// Mitsubishi GX Works2 project: projectfinalahushiling   PLC: FX3G

// global labels: Global1
VAR_GLOBAL
  startBaking AT X001 : BOOL;
  bakingTimer AT TC6 : BOOL;
END_VAR
VAR_GLOBAL CONSTANT
  bakingSec : INT := 40;
END_VAR
VAR_GLOBAL
  endBaking AT TS6 : BOOL;
  bakingLamp AT Y004 : BOOL;
  endBakingP AT M9 : BOOL;
  startBakingTimer AT TS6 : BOOL;
  endBakingTimer AT TS6 : BOOL;
  startDay AT X010 : BOOL;
  checkStock AT M0 : BOOL;
  workDayOn AT Y010 : BOOL;
  emergancyButton AT X007 : BOOL;
  validStock AT M1 : BOOL;
  flourStock AT D1100 : REAL;
END_VAR
VAR_GLOBAL CONSTANT
  flourInit : REAL := 100;
END_VAR
VAR_GLOBAL
  flour_input AT D1150 : REAL;
  yeast_input AT D1152 : REAL;
  oil_input AT D1154 : REAL;
  water_input AT D1156 : REAL;
  spieces_input AT D1158 : REAL;
  yeastStock AT D1102 : REAL;
  oilStock AT D1104 : REAL;
  waterStock AT D1106 : REAL;
  spicesStock AT D1108 : REAL;
END_VAR
VAR_GLOBAL CONSTANT
  ratioYeast : REAL := 2.0;
  ratioOil : REAL := 3.0;
  waterRatio : REAL := 5.0;
  spicesRatio : REAL := 1.0;
  times10 : REAL := 10.0;
END_VAR
VAR_GLOBAL
  yeastTimes10 AT D1110 : REAL;
  oilTimes10 AT D1112 : REAL;
  waterTimes10 AT D1114 : REAL;
  spicesTimes10 AT D1116 : REAL;
  flourTimesYeast AT D1118 : REAL;
  flourTimesOil AT D1120 : REAL;
  flourTimesWater AT D1122 : REAL;
  flourTimesSpices AT D1124 : REAL;
  startPrep AT X002 : BOOL;
  EndPrep AT TS1 : BOOL;
  LampPrep AT Y005 : BOOL;
  timeForPrep AT TC1 : BOOL;
END_VAR
VAR_GLOBAL CONSTANT
  secondsPrep : INT := 30;
END_VAR
VAR_GLOBAL
  PrepDone AT M5 : BOOL;
END_VAR
VAR_GLOBAL CONSTANT
  yeastNeed : REAL := 20.0;
  waterNeed : REAL := 50;
  OilNeed : REAL := 30.0;
  spiceNeed : REAL := 10;
END_VAR
VAR_GLOBAL
  flourInMixer AT D1130 : REAL;
  YeastrInMixer AT D1132 : REAL;
  waterInMixer AT D1134 : REAL;
  oilInMixer AT D1136 : REAL;
  spiceInMixer AT D1138 : REAL;
  endMix AT M2 : BOOL;
  endMix2 AT M23 : BOOL;
  endMix3 AT M24 : BOOL;
  endMix4 AT M25 : BOOL;
  endMix5 AT M26 : BOOL;
  startLisha AT X001 : BOOL;
  endCountPressings AT CS0 : BOOL;
  lishaLamp AT Y001 : BOOL;
  flourInLisha AT D1140 : REAL;
  YeastrInLish AT D1142 : REAL;
  waterInLisha AT D1144 : REAL;
  oilInLisha AT D1146 : REAL;
  spiceInLisha AT D1148 : REAL;
  startSwelling AT X011 : BOOL;
END_VAR
VAR_GLOBAL CONSTANT
  doublePressings : INT := 2;
END_VAR
VAR_GLOBAL
  countPressings AT CC0 : BOOL;
  flourInProofing AT D1160 : REAL;
  YeastrInProofing AT D1162 : REAL;
  waterInProofing AT D1164 : REAL;
  oilInProofing AT D1166 : REAL;
  spiceInProofing AT D1168 : REAL;
  helpLight AT M3 : BOOL;
  flinckering2 AT Y003 : BOOL;
  flinckering1 AT Y002 : BOOL;
  TC_2 AT TC2 : BOOL;
END_VAR
VAR_GLOBAL CONSTANT
  OnOff : INT := 30;
END_VAR
VAR_GLOBAL
  TC_3 AT TC3 : BOOL;
  TS_3 AT TS3 : BOOL;
  TS_2 AT TS2 : BOOL;
  endLishaP AT M4 : BOOL;
  endProofingTimer AT TS4 : BOOL;
  proofingTimer AT TC4 : BOOL;
  endProofingP AT M4 : BOOL;
  endLisha1 AT M31 : BOOL;
  TS_4 AT TS4 : BOOL;
END_VAR
VAR_GLOBAL CONSTANT
  OnOff1 : INT := 5;
  OnOff2 : INT := 5;
END_VAR
VAR_GLOBAL
  qualityCheck AT X003 : BOOL;
  Analog_Input_2 AT D8281 : REAL;
  qualityBread AT D8201 : INT;
END_VAR
VAR_GLOBAL CONSTANT
  minQuality : INT := 400;
  maxQuality : INT := 2000;
END_VAR
VAR_GLOBAL
  startProofing AT M4 : BOOL;
  flourInBake AT D1190 : REAL;
  flourInProofingflourInBake AT D1190 : REAL;
  YeastrInBake AT D1192 : REAL;
  waterInBake AT D1194 : REAL;
  OilInBake AT D1196 : REAL;
  spiceInBake AT D1198 : REAL;
  noHaveStock AT M20 : BOOL;
  counterAnswer AT CS2 : BOOL;
  D_8281 AT D8281 : INT;
  checkCount AT CC2 : BOOL;
END_VAR
VAR_GLOBAL CONSTANT
  twoChecks : INT := 2;
END_VAR
VAR_GLOBAL
  lowThan AT M17 : BOOL;
  greaterThan AT M18 : BOOL;
  qualityCheckGood AT M11 : BOOL;
  breadReadyTimer AT TC8 : BOOL;
END_VAR
VAR_GLOBAL CONSTANT
  readyTime : INT := 50;
END_VAR
VAR_GLOBAL
  endFinishTimer AT TS8 : BOOL;
  finishLamp AT Y006 : BOOL;
  breadInBaking AT D7500 : REAL;
  breadToBakery AT D7700 : REAL;
END_VAR
VAR_GLOBAL CONSTANT
  reset : REAL;
END_VAR
VAR_GLOBAL
  dayOver AT M100 : BOOL;
  resetIngridiens AT M35 : BOOL;
  flag AT M40 : BOOL;
  Pulse AT M5 : BOOL;
  checkC AT M41 : BOOL;
  Try AT M101 : BOOL;
  reset12 AT M35 : BOOL;
  resetTry AT M50 : BOOL;
  finishLampPrep AT Y006 : BOOL;
  notEnoughIng AT M67 : BOOL;
  finishIteration AT M120 : BOOL;
  finishIteration2 AT M122 : BOOL;
  finishDay AT M20 : BOOL;
  M_51 AT M51 : BOOL;
  M_11 AT M111 : BOOL;
  M_52 AT M52 : BOOL;
  emergency AT X007 : BOOL;
  TC_7 AT TC7 : BOOL;
  TS_7 AT TS7 : BOOL;
  M_30 AT M30 : BOOL;
  TC_10 AT TC10 : BOOL;
END_VAR
VAR_GLOBAL CONSTANT
  const5 : INT := 5;
END_VAR
VAR_GLOBAL
  TS_10 AT TS10 : BOOL;
  M_12 AT M12 : BOOL;
END_VAR
VAR_GLOBAL CONSTANT
  sec3 : INT := 30;
END_VAR
VAR_GLOBAL
  TC_11 AT TC11 : BOOL;
  TS_11 AT TS11 : BOOL;
  M_111 AT M111 : BOOL;
  finishDayLight AT M20 : BOOL;
END_VAR
VAR_GLOBAL CONSTANT
  flourInit1 : REAL := 99;
END_VAR

// task Task_01 (event TRUE, interval 0, priority 31): POU_01

PROGRAM POU_01
(* structured ladder/FBD written out as ST: instructions are called as NAME(EN, inputs, outputs); _pN, _eN, _tN stand for wires *)
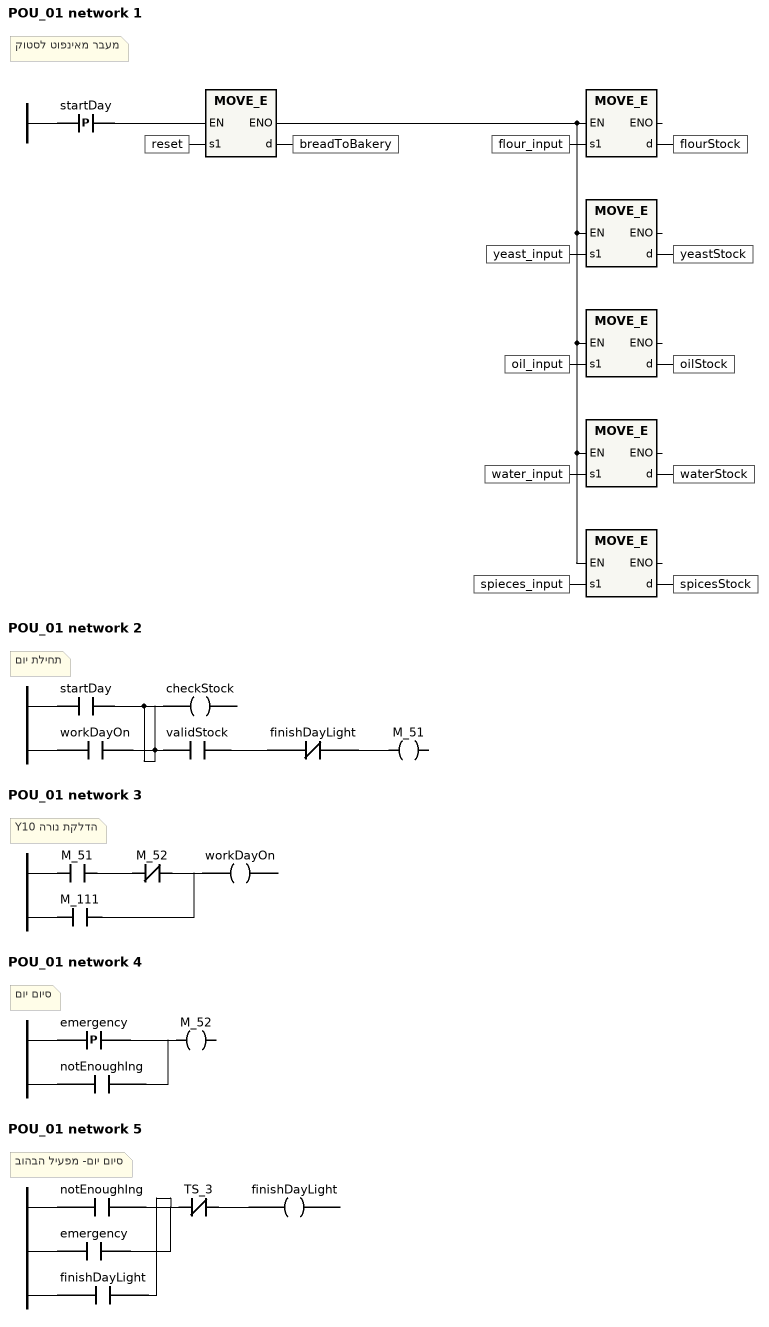
(* network 1 *)
(* מעבר מאינפוט לסטוק *)
_e1 := MOVE_E(LDP(TRUE, startDay), reset, breadToBakery);
MOVE_E(_e1, flour_input, flourStock);
MOVE_E(_e1, yeast_input, yeastStock);
MOVE_E(_e1, oil_input, oilStock);
MOVE_E(_e1, water_input, waterStock);
MOVE_E(_e1, spieces_input, spicesStock);
(* network 2 *)
(* תחילת יום *)
_p1 := startDay OR workDayOn;
checkStock := _p1;
M_51 := _p1 AND validStock AND NOT finishDayLight;
(* network 3 *)
(* הדלקת נורה Y10 *)
workDayOn := (M_51 AND NOT M_52) OR M_111;
(* network 4 *)
(* סיום יום *)
M_52 := LDP(TRUE, emergency) OR notEnoughIng;
(* network 5 *)
(* סיום יום- מפעיל הבהוב *)
finishDayLight := (notEnoughIng OR emergency OR finishDayLight) AND NOT TS_3;
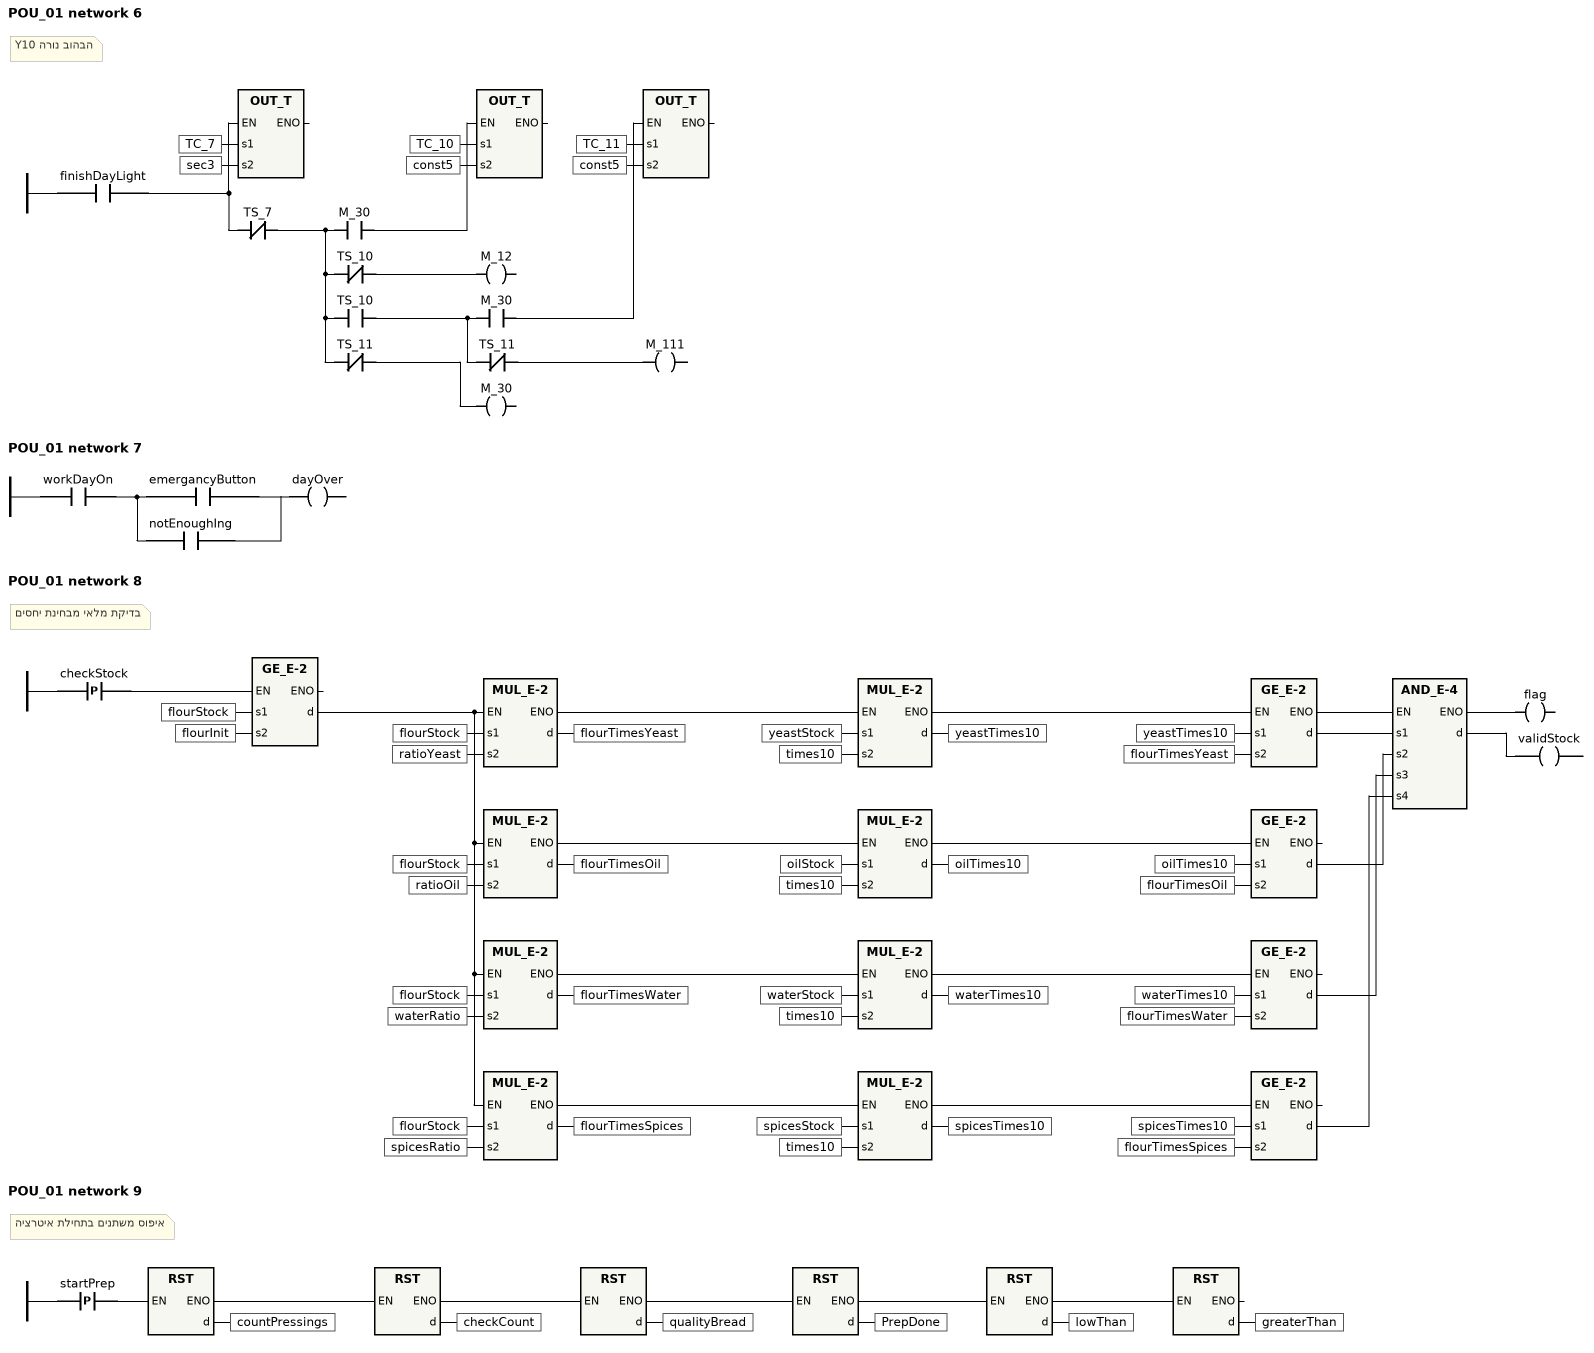
(* network 6 *)
(* הבהוב נורה Y10 *)
OUT_T(finishDayLight, TC_7, sec3);
_p1 := finishDayLight AND NOT TS_7;
OUT_T(_p1 AND M_30, TC_10, const5);
M_12 := _p1 AND NOT TS_10;
_p2 := _p1 AND TS_10;
OUT_T(_p2 AND M_30, TC_11, const5);
M_111 := _p2 AND NOT TS_11;
M_30 := _p1 AND NOT TS_11;
(* network 7 *)
dayOver := (workDayOn AND emergancyButton) OR (workDayOn AND notEnoughIng);
(* network 8 *)
(* בדיקת מלאי מבחינת יחסים *)
GE_E(LDP(TRUE, checkStock), flourStock, flourInit, _t1);
_e2 := MUL_E(_t1, flourStock, ratioYeast, flourTimesYeast);
_e3 := MUL_E(_e2, yeastStock, times10, yeastTimes10);
_e5 := GE_E(_e3, yeastTimes10, flourTimesYeast, _t4);
_e6 := MUL_E(_t1, flourStock, ratioOil, flourTimesOil);
_e7 := MUL_E(_e6, oilStock, times10, oilTimes10);
GE_E(_e7, oilTimes10, flourTimesOil, _t8);
_e9 := MUL_E(_t1, flourStock, waterRatio, flourTimesWater);
_e10 := MUL_E(_e9, waterStock, times10, waterTimes10);
GE_E(_e10, waterTimes10, flourTimesWater, _t11);
_e12 := MUL_E(_t1, flourStock, spicesRatio, flourTimesSpices);
_e13 := MUL_E(_e12, spicesStock, times10, spicesTimes10);
GE_E(_e13, spicesTimes10, flourTimesSpices, _t14);
_e16 := AND_E(_e5, _t4, _t8, _t11, _t14, _t15);
flag := _e16;
validStock := _t15;
(* network 9 *)
(* איפוס משתנים בתחילת איטרציה *)
_e1 := RST(LDP(TRUE, startPrep), countPressings);
_e2 := RST(_e1, checkCount);
_e3 := RST(_e2, qualityBread);
_e4 := RST(_e3, PrepDone);
_e5 := RST(_e4, lowThan);
RST(_e5, greaterThan);
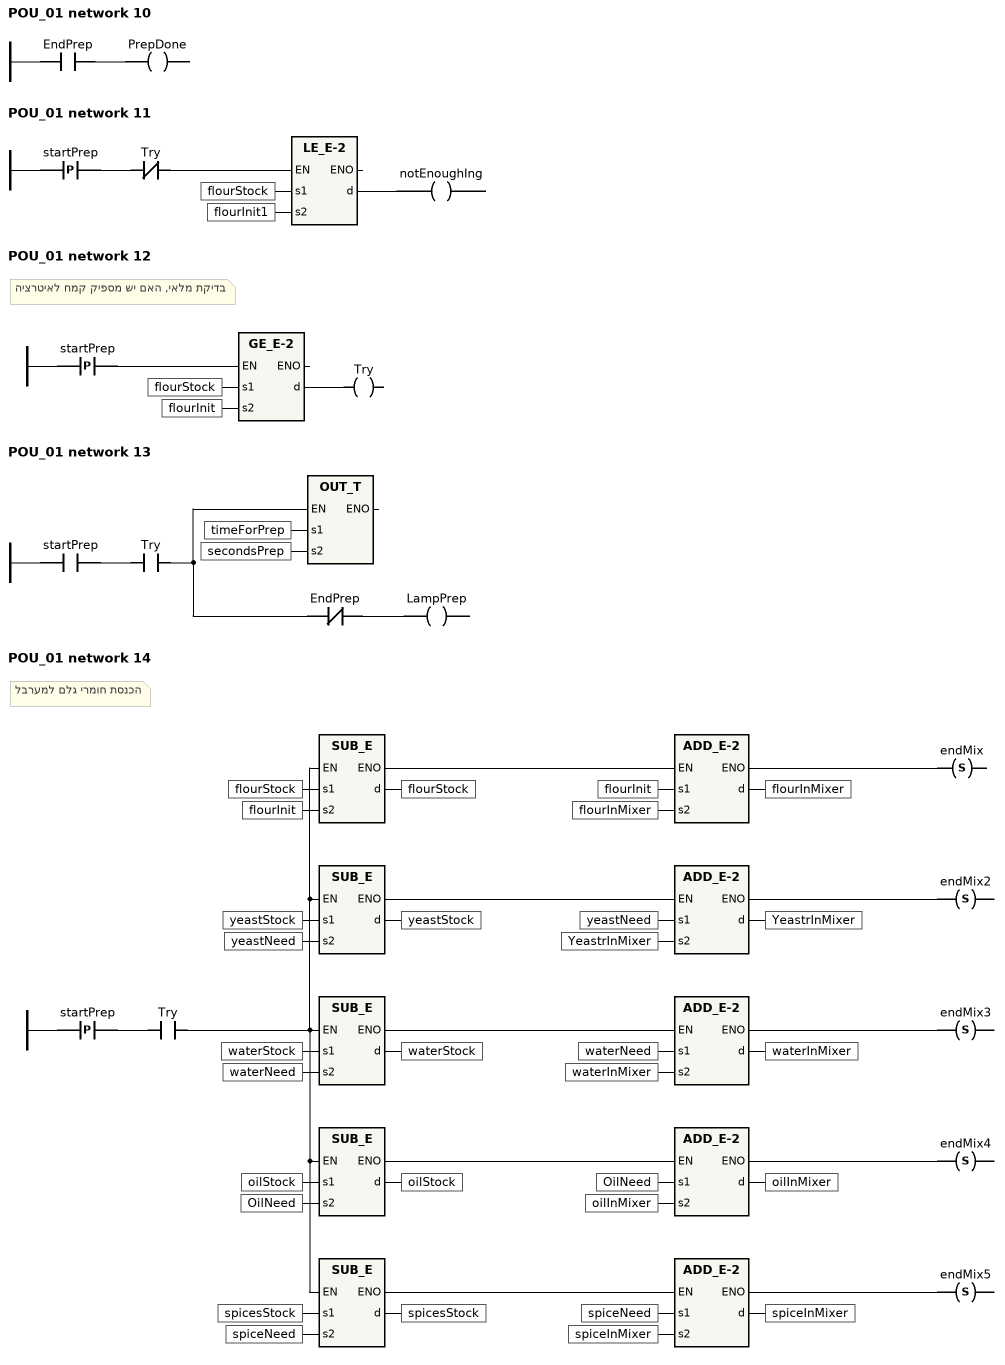
(* network 10 *)
PrepDone := EndPrep;
(* network 11 *)
LE_E(LDP(TRUE, startPrep) AND NOT Try, flourStock, flourInit1, _t1);
notEnoughIng := _t1;
(* network 12 *)
(* בדיקת מלאי, האם יש מספיק קמח לאיטרציה *)
GE_E(LDP(TRUE, startPrep), flourStock, flourInit, _t1);
Try := _t1;
(* network 13 *)
_p1 := startPrep AND Try;
OUT_T(_p1, timeForPrep, secondsPrep);
LampPrep := _p1 AND NOT EndPrep;
(* network 14 *)
(* הכנסת חומרי גלם למערבל *)
_p1 := LDP(TRUE, startPrep) AND Try;
_e2 := SUB_E(_p1, flourStock, flourInit, flourStock);
_e3 := ADD_E(_e2, flourInit, flourInMixer, flourInMixer);
SET(_e3, endMix);
_e4 := SUB_E(_p1, yeastStock, yeastNeed, yeastStock);
_e5 := ADD_E(_e4, yeastNeed, YeastrInMixer, YeastrInMixer);
SET(_e5, endMix2);
_e6 := SUB_E(_p1, waterStock, waterNeed, waterStock);
_e7 := ADD_E(_e6, waterNeed, waterInMixer, waterInMixer);
SET(_e7, endMix3);
_e8 := SUB_E(_p1, oilStock, OilNeed, oilStock);
_e9 := ADD_E(_e8, OilNeed, oilInMixer, oilInMixer);
SET(_e9, endMix4);
_e10 := SUB_E(_p1, spicesStock, spiceNeed, spicesStock);
_e11 := ADD_E(_e10, spiceNeed, spiceInMixer, spiceInMixer);
SET(_e11, endMix5);
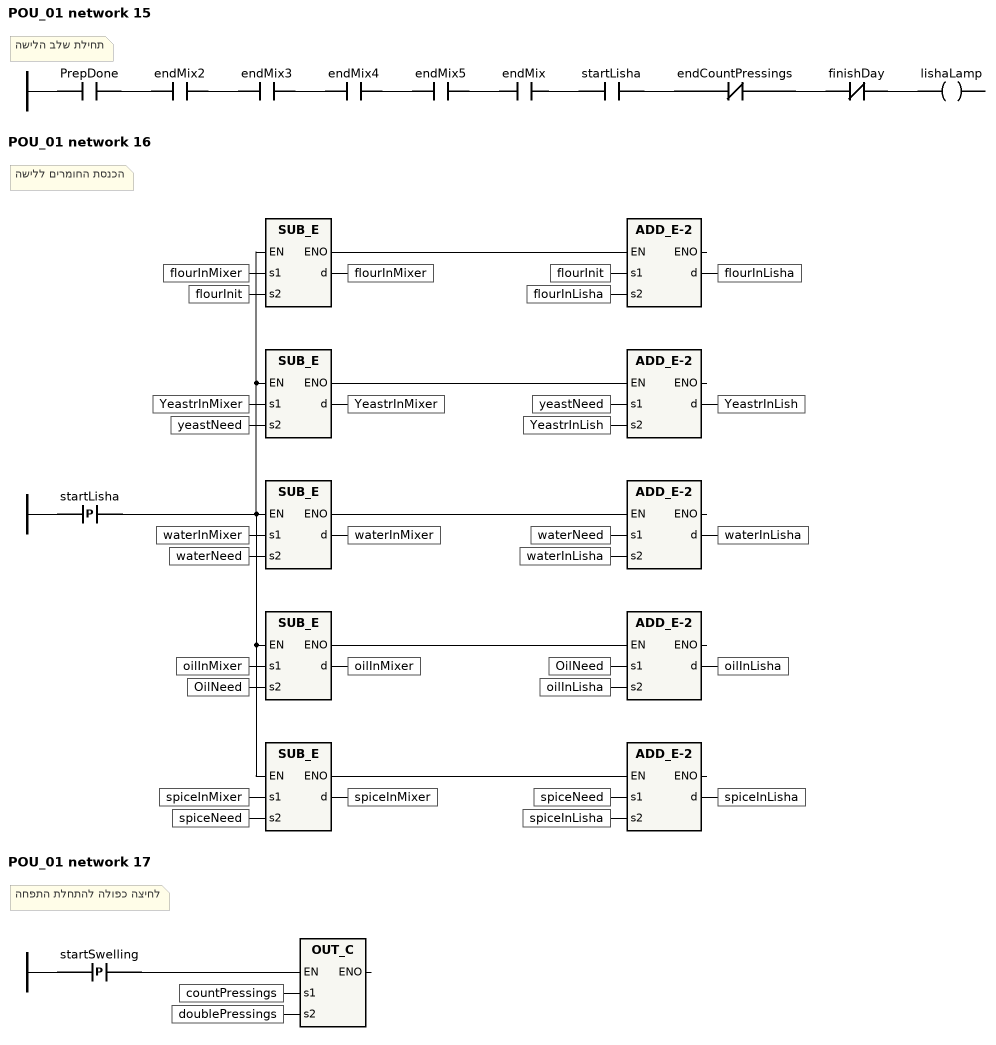
(* network 15 *)
(* תחילת שלב הלישה *)
lishaLamp := PrepDone AND endMix2 AND endMix3 AND endMix4 AND endMix5 AND endMix AND startLisha AND NOT endCountPressings AND NOT finishDay;
(* network 16 *)
(* הכנסת החומרים ללישה *)
_p1 := LDP(TRUE, startLisha);
_e2 := SUB_E(_p1, flourInMixer, flourInit, flourInMixer);
ADD_E(_e2, flourInit, flourInLisha, flourInLisha);
_e3 := SUB_E(_p1, YeastrInMixer, yeastNeed, YeastrInMixer);
ADD_E(_e3, yeastNeed, YeastrInLish, YeastrInLish);
_e4 := SUB_E(_p1, waterInMixer, waterNeed, waterInMixer);
ADD_E(_e4, waterNeed, waterInLisha, waterInLisha);
_e5 := SUB_E(_p1, oilInMixer, OilNeed, oilInMixer);
ADD_E(_e5, OilNeed, oilInLisha, oilInLisha);
_e6 := SUB_E(_p1, spiceInMixer, spiceNeed, spiceInMixer);
ADD_E(_e6, spiceNeed, spiceInLisha, spiceInLisha);
(* network 17 *)
(* לחיצה כפולה להתחלת התפחה *)
OUT_C(LDP(TRUE, startSwelling), countPressings, doublePressings);
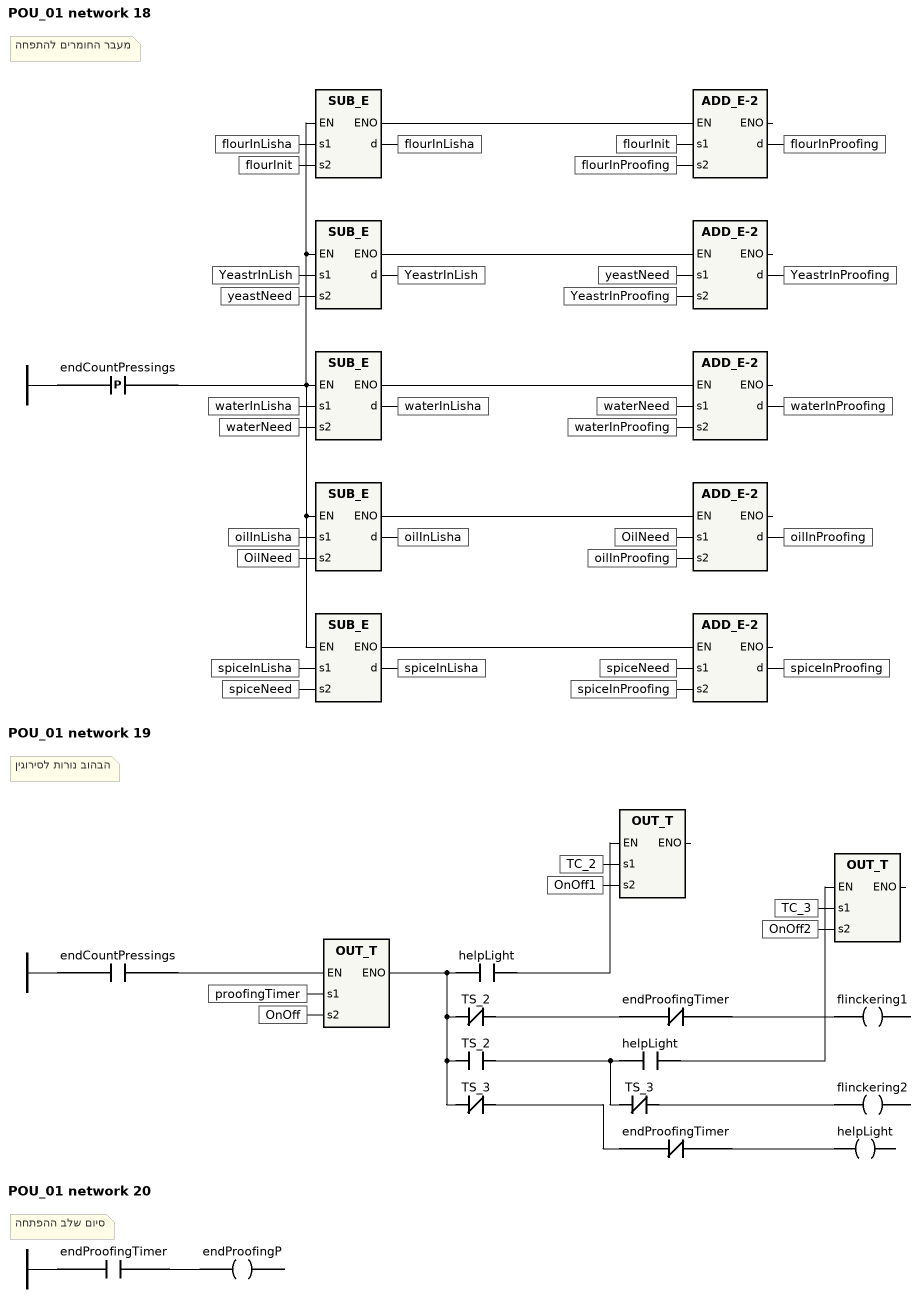
(* network 18 *)
(* מעבר החומרים להתפחה *)
_p1 := LDP(TRUE, endCountPressings);
_e2 := SUB_E(_p1, flourInLisha, flourInit, flourInLisha);
ADD_E(_e2, flourInit, flourInProofing, flourInProofing);
_e3 := SUB_E(_p1, YeastrInLish, yeastNeed, YeastrInLish);
ADD_E(_e3, yeastNeed, YeastrInProofing, YeastrInProofing);
_e4 := SUB_E(_p1, waterInLisha, waterNeed, waterInLisha);
ADD_E(_e4, waterNeed, waterInProofing, waterInProofing);
_e5 := SUB_E(_p1, oilInLisha, OilNeed, oilInLisha);
ADD_E(_e5, OilNeed, oilInProofing, oilInProofing);
_e6 := SUB_E(_p1, spiceInLisha, spiceNeed, spiceInLisha);
ADD_E(_e6, spiceNeed, spiceInProofing, spiceInProofing);
(* network 19 *)
(* הבהוב נורות לסירוגין *)
_e1 := OUT_T(endCountPressings, proofingTimer, OnOff);
OUT_T(_e1 AND helpLight, TC_2, OnOff1);
flinckering1 := _e1 AND NOT TS_2 AND NOT endProofingTimer;
_p2 := _e1 AND TS_2;
OUT_T(_p2 AND helpLight, TC_3, OnOff2);
flinckering2 := _p2 AND NOT TS_3;
helpLight := _e1 AND NOT TS_3 AND NOT endProofingTimer;
(* network 20 *)
(* סיום שלב ההפתחה *)
endProofingP := endProofingTimer;
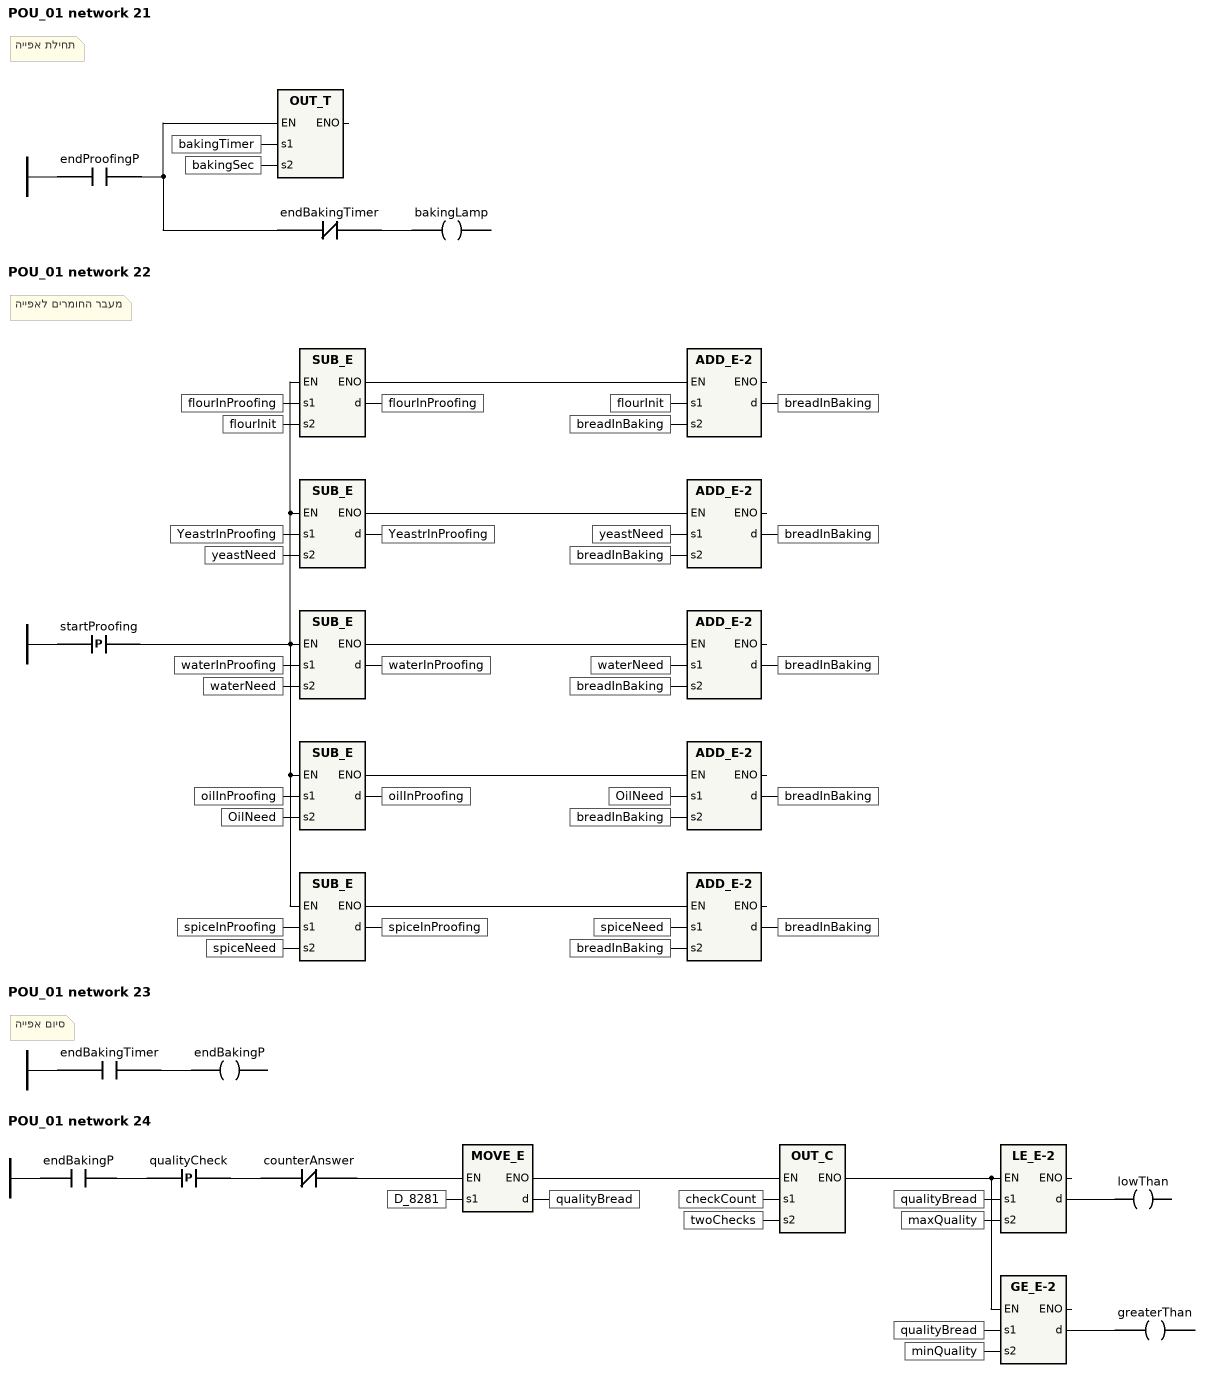
(* network 21 *)
(* תחילת אפייה *)
OUT_T(endProofingP, bakingTimer, bakingSec);
bakingLamp := endProofingP AND NOT endBakingTimer;
(* network 22 *)
(* מעבר החומרים לאפייה *)
_p1 := LDP(TRUE, startProofing);
_e2 := SUB_E(_p1, flourInProofing, flourInit, flourInProofing);
ADD_E(_e2, flourInit, breadInBaking, breadInBaking);
_e3 := SUB_E(_p1, YeastrInProofing, yeastNeed, YeastrInProofing);
ADD_E(_e3, yeastNeed, breadInBaking, breadInBaking);
_e4 := SUB_E(_p1, waterInProofing, waterNeed, waterInProofing);
ADD_E(_e4, waterNeed, breadInBaking, breadInBaking);
_e5 := SUB_E(_p1, oilInProofing, OilNeed, oilInProofing);
ADD_E(_e5, OilNeed, breadInBaking, breadInBaking);
_e6 := SUB_E(_p1, spiceInProofing, spiceNeed, spiceInProofing);
ADD_E(_e6, spiceNeed, breadInBaking, breadInBaking);
(* network 23 *)
(* סיום אפייה *)
endBakingP := endBakingTimer;
(* network 24 *)
_e1 := MOVE_E(endBakingP AND LDP(TRUE, qualityCheck) AND NOT counterAnswer, D_8281, qualityBread);
_e2 := OUT_C(_e1, checkCount, twoChecks);
LE_E(_e2, qualityBread, maxQuality, _t3);
lowThan := _t3;
GE_E(_e2, qualityBread, minQuality, _t4);
greaterThan := _t4;
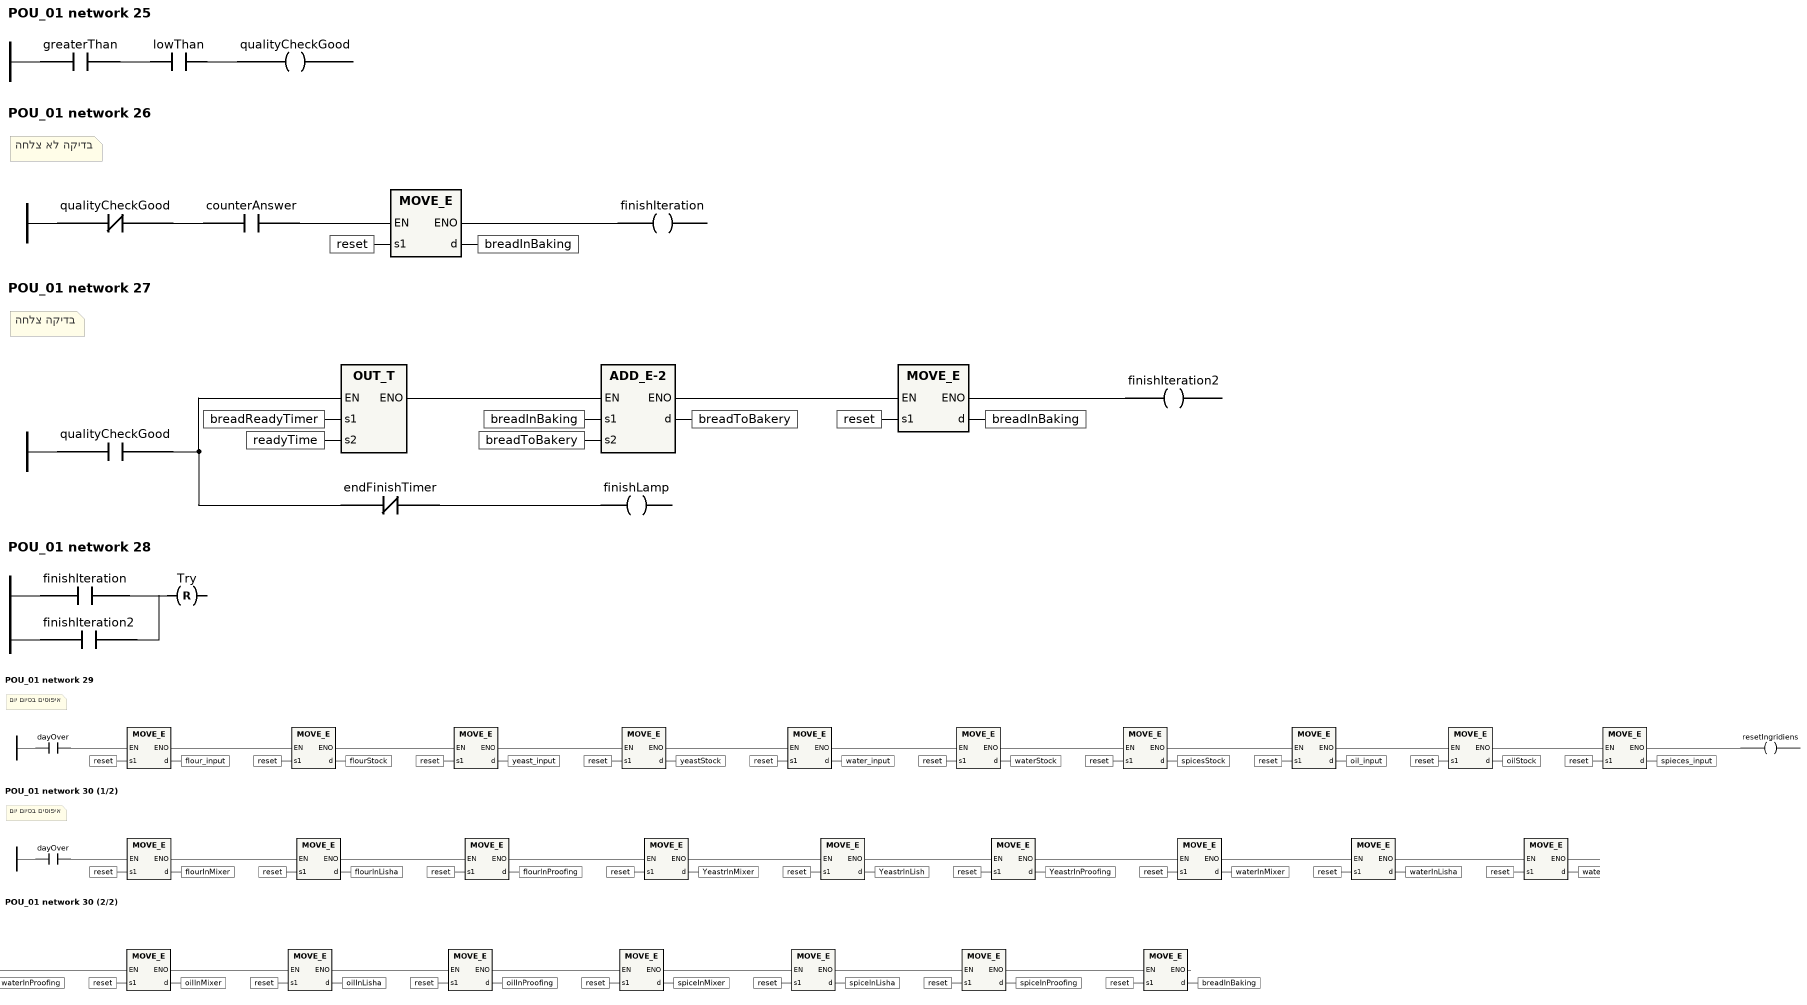
(* network 25 *)
qualityCheckGood := greaterThan AND lowThan;
(* network 26 *)
(* בדיקה לא צלחה *)
_e1 := MOVE_E(NOT qualityCheckGood AND counterAnswer, reset, breadInBaking);
finishIteration := _e1;
(* network 27 *)
(* בדיקה צלחה *)
_e1 := OUT_T(qualityCheckGood, breadReadyTimer, readyTime);
_e2 := ADD_E(_e1, breadInBaking, breadToBakery, breadToBakery);
_e3 := MOVE_E(_e2, reset, breadInBaking);
finishIteration2 := _e3;
finishLamp := qualityCheckGood AND NOT endFinishTimer;
(* network 28 *)
RST(finishIteration OR finishIteration2, Try);
(* network 29 *)
(* איפוסים בסיום יום *)
_e1 := MOVE_E(dayOver, reset, flour_input);
_e2 := MOVE_E(_e1, reset, flourStock);
_e3 := MOVE_E(_e2, reset, yeast_input);
_e4 := MOVE_E(_e3, reset, yeastStock);
_e5 := MOVE_E(_e4, reset, water_input);
_e6 := MOVE_E(_e5, reset, waterStock);
_e7 := MOVE_E(_e6, reset, spicesStock);
_e8 := MOVE_E(_e7, reset, oil_input);
_e9 := MOVE_E(_e8, reset, oilStock);
_e10 := MOVE_E(_e9, reset, spieces_input);
resetIngridiens := _e10;
(* network 30 *)
(* איפוסים בסיום יום *)
_e1 := MOVE_E(dayOver, reset, flourInMixer);
_e2 := MOVE_E(_e1, reset, flourInLisha);
_e3 := MOVE_E(_e2, reset, flourInProofing);
_e4 := MOVE_E(_e3, reset, YeastrInMixer);
_e5 := MOVE_E(_e4, reset, YeastrInLish);
_e6 := MOVE_E(_e5, reset, YeastrInProofing);
_e7 := MOVE_E(_e6, reset, waterInMixer);
_e8 := MOVE_E(_e7, reset, waterInLisha);
_e9 := MOVE_E(_e8, reset, waterInProofing);
_e10 := MOVE_E(_e9, reset, oilInMixer);
_e11 := MOVE_E(_e10, reset, oilInLisha);
_e12 := MOVE_E(_e11, reset, oilInProofing);
_e13 := MOVE_E(_e12, reset, spiceInMixer);
_e14 := MOVE_E(_e13, reset, spiceInLisha);
_e15 := MOVE_E(_e14, reset, spiceInProofing);
MOVE_E(_e15, reset, breadInBaking);
END_PROGRAM
